{attribute 'Tc2GvlVarNames'}
VAR_CONFIG
END_VAR

(* stored: Version 1.1.0.1, ProductVersion 3.1.4024.5
   GVL Variable_Configuration: Id {d0fb6070-f344-42f4-9b9a-b30d23963261} *)
